// TIA Portal V21 export
TYPE "Std_SendReceive"
   STRUCT
      Digitali : Array[0..31] of "Std_Segnale";
      "DInt" : Array[0..19] of DInt;
      "Real" : Array[0..19] of Real;
      Prm : Struct
         Abilitazione : Bool;   // Abilitazione alla lettura o scrittura
      END_STRUCT;
   END_STRUCT;
   // // Digitali[0] : Watchdog
   // // "DInt"[0] : Watchdog
END_TYPE
